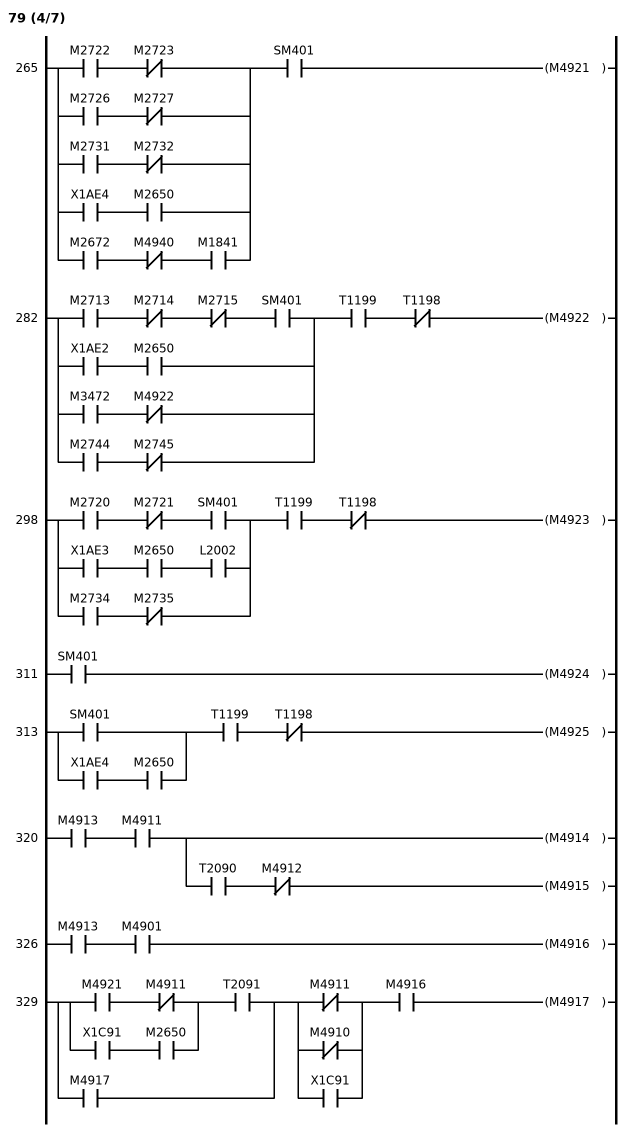
265   LD      M2722
      ANI     M2723
      LD      M2726
      ANI     M2727
      ORB
      LD      M2731
      ANI     M2732
      ORB
      LD      X1AE4
      AND     M2650
      ORB
      LD      M2672
      ANI     M4940
      AND     M1841
      ORB
      AND     SM401
      OUT     M4921
282   LD      M2713
      ANI     M2714
      ANI     M2715
      AND     SM401
      LD      X1AE2
      AND     M2650
      ORB
      LD      M3472
      ANI     M4922
      ORB
      LD      M2744
      ANI     M2745
      ORB
      AND     T1199
      ANI     T1198
      OUT     M4922
298   LD      M2720
      ANI     M2721
      AND     SM401
      LD      X1AE3
      AND     M2650
      AND     L2002
      ORB
      LD      M2734
      ANI     M2735
      ORB
      AND     T1199
      ANI     T1198
      OUT     M4923
311   LD      SM401
      OUT     M4924
313   LD      SM401
      LD      X1AE4
      AND     M2650
      ORB
      AND     T1199
      ANI     T1198
      OUT     M4925
320   LD      M4913
      AND     M4911
      OUT     M4914
      AND     T2090
      ANI     M4912
      OUT     M4915
326   LD      M4913
      AND     M4901
      OUT     M4916
329   LD      M4921
      ANI     M4911
      LD      X1C91
      AND     M2650
      ORB
      AND     T2091
      OR      M4917
      LDI     M4911
      ORI     M4910
      OR      X1C91
      ANB
      AND     M4916
      OUT     M4917
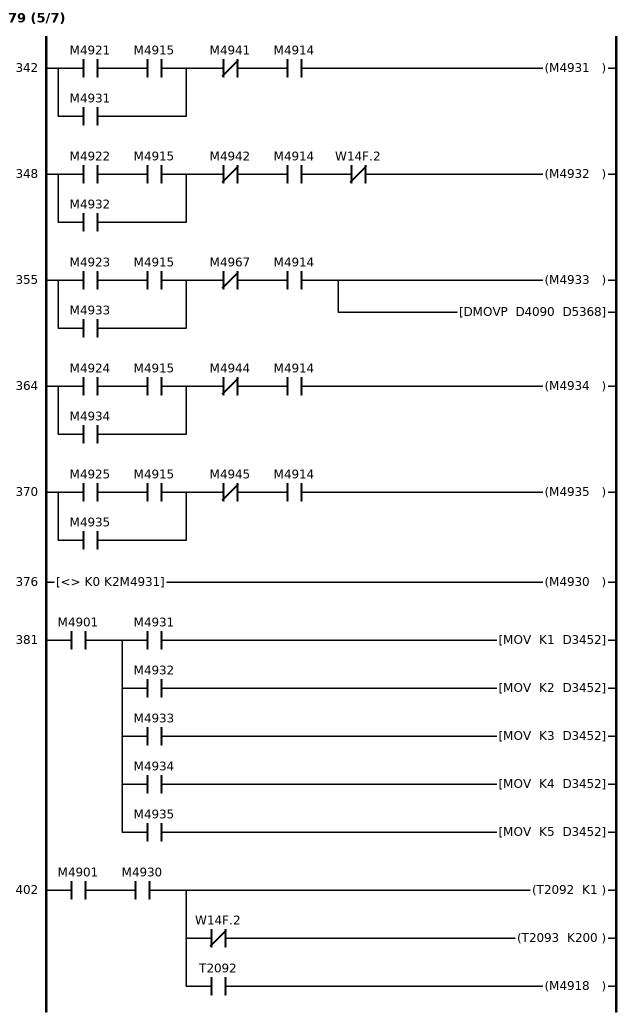
342   LD      M4921
      AND     M4915
      OR      M4931
      ANI     M4941
      AND     M4914
      OUT     M4931
348   LD      M4922
      AND     M4915
      OR      M4932
      ANI     M4942
      AND     M4914
      ANI     W14F.2
      OUT     M4932
355   LD      M4923
      AND     M4915
      OR      M4933
      ANI     M4967
      AND     M4914
      OUT     M4933
      DMOVP   D4090 D5368
364   LD      M4924
      AND     M4915
      OR      M4934
      ANI     M4944
      AND     M4914
      OUT     M4934
370   LD      M4925
      AND     M4915
      OR      M4935
      ANI     M4945
      AND     M4914
      OUT     M4935
376   LD<>    K0 K2M4931
      OUT     M4930
381   LD      M4901
      MPS
      AND     M4931
      MOV     K1 D3452
      MRD
      AND     M4932
      MOV     K2 D3452
      MRD
      AND     M4933
      MOV     K3 D3452
      MRD
      AND     M4934
      MOV     K4 D3452
      MPP
      AND     M4935
      MOV     K5 D3452
402   LD      M4901
      AND     M4930
      OUT     T2092 K1
      MPS
      ANI     W14F.2
      OUT     T2093 K200
      MPP
      AND     T2092
      OUT     M4918
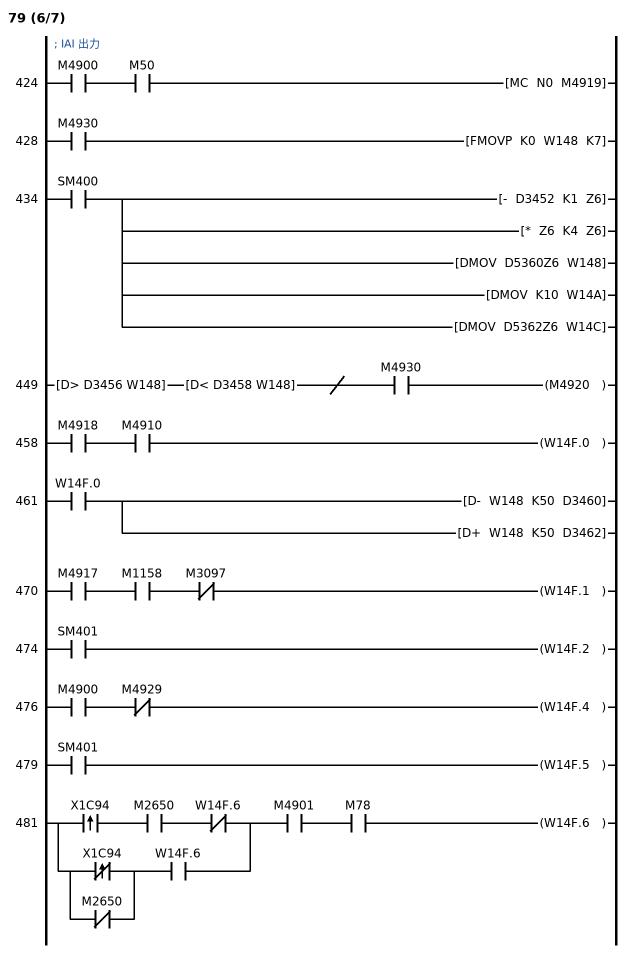
; IAI 出力
424   LD      M4900
      AND     M50
      MC      N0 M4919
428   LD      M4930
      FMOVP   K0 W148 K7
434   LD      SM400
      -       D3452 K1 Z6
      *       Z6 K4 Z6
      DMOV    D5360Z6 W148
      DMOV    K10 W14A
      DMOV    D5362Z6 W14C
449   LDD>    D3456 W148
      ANDD<   D3458 W148
      INV
      AND     M4930
      OUT     M4920
458   LD      M4918
      AND     M4910
      OUT     W14F.0
461   LD      W14F.0
      D-      W148 K50 D3460
      D+      W148 K50 D3462
470   LD      M4917
      AND     M1158
      ANI     M3097
      OUT     W14F.1
474   LD      SM401
      OUT     W14F.2
476   LD      M4900
      ANI     M4929
      OUT     W14F.4
479   LD      SM401
      OUT     W14F.5
481   LDP     X1C94
      AND     M2650
      ANI     W14F.6
      LDPI    X1C94
      ORI     M2650
      AND     W14F.6
      ORB
      AND     M4901
      AND     M78
      OUT     W14F.6
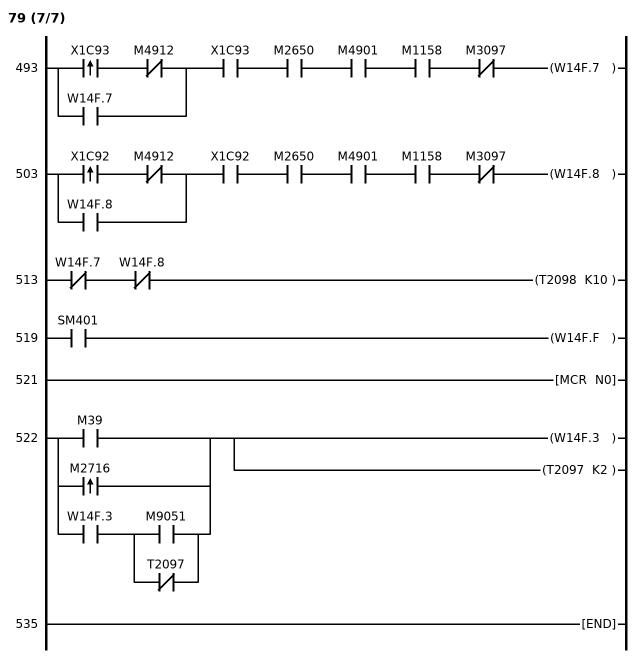
493   LDP     X1C93
      ANI     M4912
      OR      W14F.7
      AND     X1C93
      AND     M2650
      AND     M4901
      AND     M1158
      ANI     M3097
      OUT     W14F.7
503   LDP     X1C92
      ANI     M4912
      OR      W14F.8
      AND     X1C92
      AND     M2650
      AND     M4901
      AND     M1158
      ANI     M3097
      OUT     W14F.8
513   LDI     W14F.7
      ANI     W14F.8
      OUT     T2098 K10
519   LD      SM401
      OUT     W14F.F
521   MCR     N0
522   LD      M39
      ORP     M2716
      LD      W14F.3
      LD      M9051
      ORI     T2097
      ANB
      ORB
      OUT     W14F.3
      OUT     T2097 K2
535   END
END_PROGRAM

PROGRAM 80
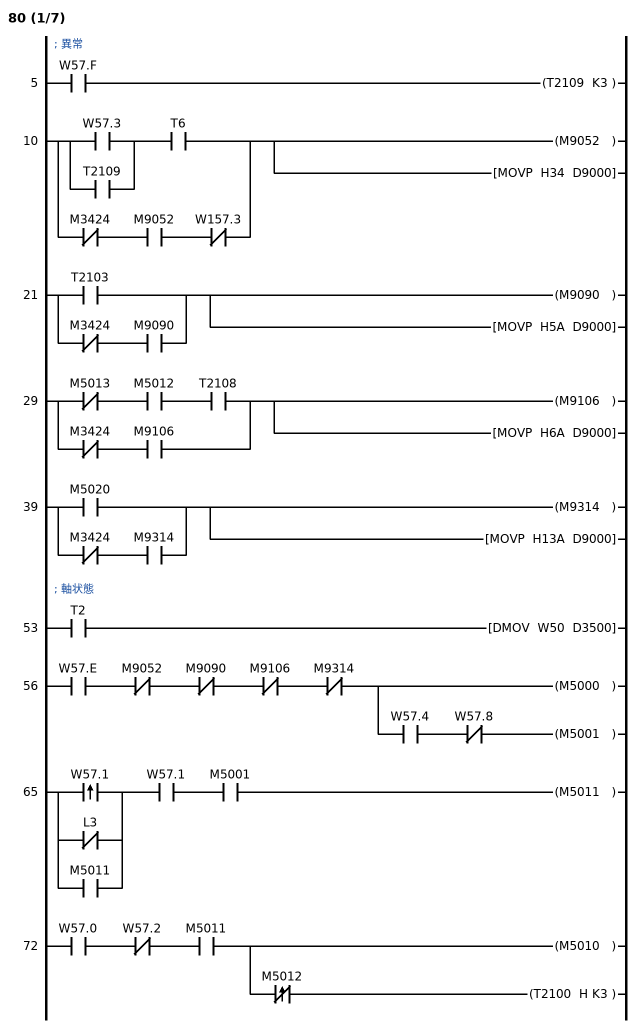
; 異常
5     LD      W57.F
      OUT     T2109 K3
10    LD      W57.3
      OR      T2109
      AND     T6
      LDI     M3424
      AND     M9052
      ANI     W157.3
      ORB
      OUT     M9052
      MOVP    H34 D9000
21    LD      T2103
      LDI     M3424
      AND     M9090
      ORB
      OUT     M9090
      MOVP    H5A D9000
29    LDI     M5013
      AND     M5012
      AND     T2108
      LDI     M3424
      AND     M9106
      ORB
      OUT     M9106
      MOVP    H6A D9000
39    LD      M5020
      LDI     M3424
      AND     M9314
      ORB
      OUT     M9314
      MOVP    H13A D9000
; 軸状態
53    LD      T2
      DMOV    W50 D3500
56    LD      W57.E
      ANI     M9052
      ANI     M9090
      ANI     M9106
      ANI     M9314
      OUT     M5000
      AND     W57.4
      ANI     W57.8
      OUT     M5001
65    LDP     W57.1
      ORI     L3
      OR      M5011
      AND     W57.1
      AND     M5001
      OUT     M5011
72    LD      W57.0
      ANI     W57.2
      AND     M5011
      OUT     M5010
      ANDPI   M5012
      OUTH    T2100 K3
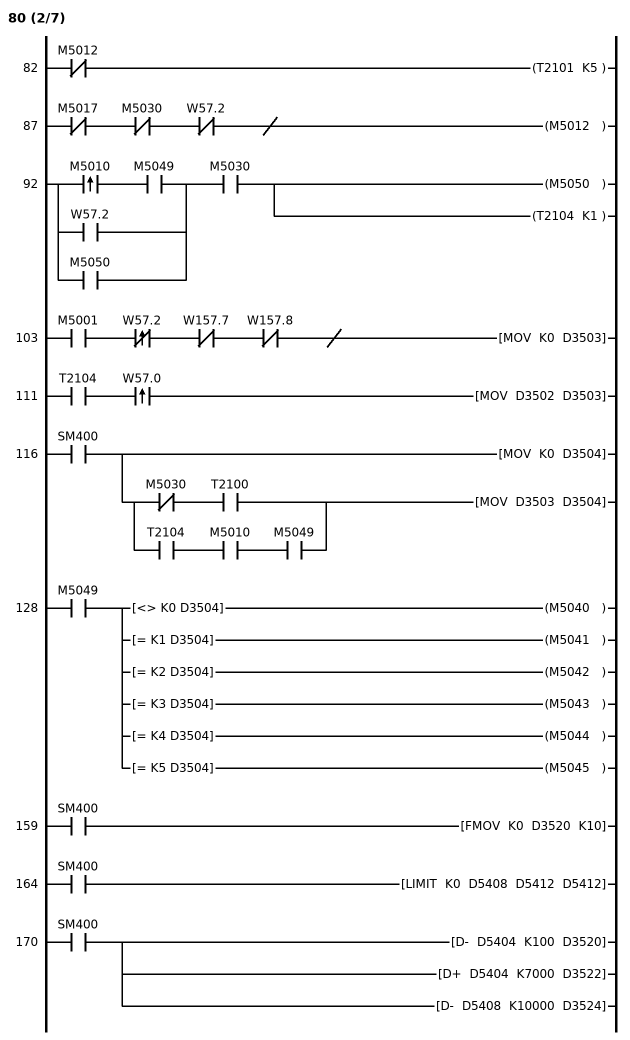
82    LDI     M5012
      OUT     T2101 K5
87    LDI     M5017
      ANI     M5030
      ANI     W57.2
      INV
      OUT     M5012
92    LDP     M5010
      AND     M5049
      OR      W57.2
      OR      M5050
      AND     M5030
      OUT     M5050
      OUT     T2104 K1
103   LD      M5001
      ANDPI   W57.2
      ANI     W157.7
      ANI     W157.8
      INV
      MOV     K0 D3503
111   LD      T2104
      ANDP    W57.0
      MOV     D3502 D3503
116   LD      SM400
      MOV     K0 D3504
      LDI     M5030
      AND     T2100
      LD      T2104
      AND     M5010
      AND     M5049
      ORB
      ANB
      MOV     D3503 D3504
128   LD      M5049
      MPS
      AND<>   K0 D3504
      OUT     M5040
      MRD
      AND=    K1 D3504
      OUT     M5041
      MRD
      AND=    K2 D3504
      OUT     M5042
      MRD
      AND=    K3 D3504
      OUT     M5043
      MRD
      AND=    K4 D3504
      OUT     M5044
      MPP
      AND=    K5 D3504
      OUT     M5045
159   LD      SM400
      FMOV    K0 D3520 K10
164   LD      SM400
      LIMIT   K0 D5408 D5412 D5412
170   LD      SM400
      D-      D5404 K100 D3520
      D+      D5404 K7000 D3522
      D-      D5408 K10000 D3524
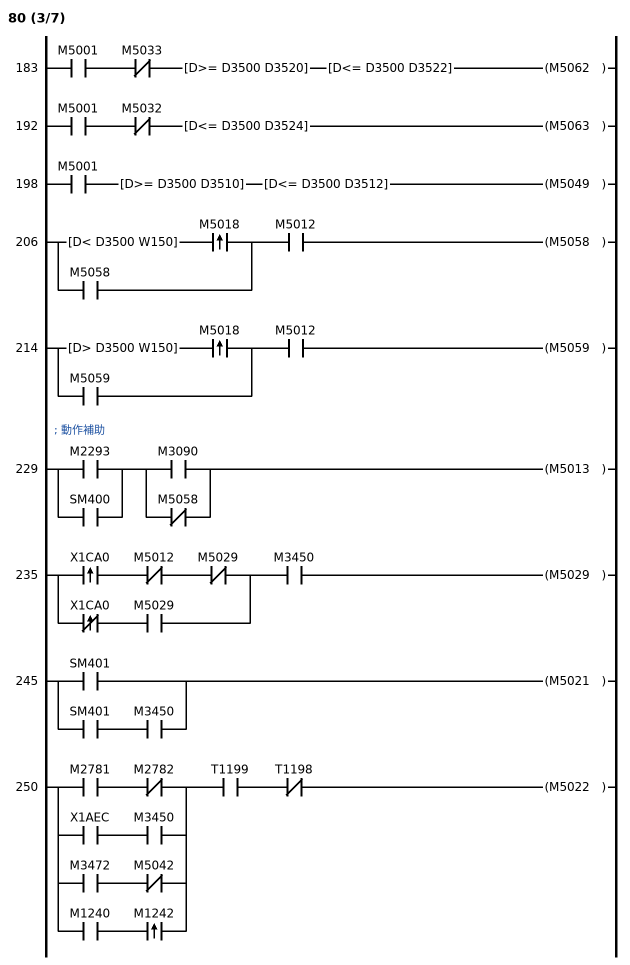
183   LD      M5001
      ANI     M5033
      ANDD>=  D3500 D3520
      ANDD<=  D3500 D3522
      OUT     M5062
192   LD      M5001
      ANI     M5032
      ANDD<=  D3500 D3524
      OUT     M5063
198   LD      M5001
      ANDD>=  D3500 D3510
      ANDD<=  D3500 D3512
      OUT     M5049
206   LDD<    D3500 W150
      ANDP    M5018
      OR      M5058
      AND     M5012
      OUT     M5058
214   LDD>    D3500 W150
      ANDP    M5018
      OR      M5059
      AND     M5012
      OUT     M5059
; 動作補助
229   LD      M2293
      OR      SM400
      LD      M3090
      ORI     M5058
      ANB
      OUT     M5013
235   LDP     X1CA0
      ANI     M5012
      ANI     M5029
      LDPI    X1CA0
      AND     M5029
      ORB
      AND     M3450
      OUT     M5029
245   LD      SM401
      LD      SM401
      AND     M3450
      ORB
      OUT     M5021
250   LD      M2781
      ANI     M2782
      LD      X1AEC
      AND     M3450
      ORB
      LD      M3472
      ANI     M5042
      ORB
      LD      M1240
      ANDP    M1242
      ORB
      AND     T1199
      ANI     T1198
      OUT     M5022
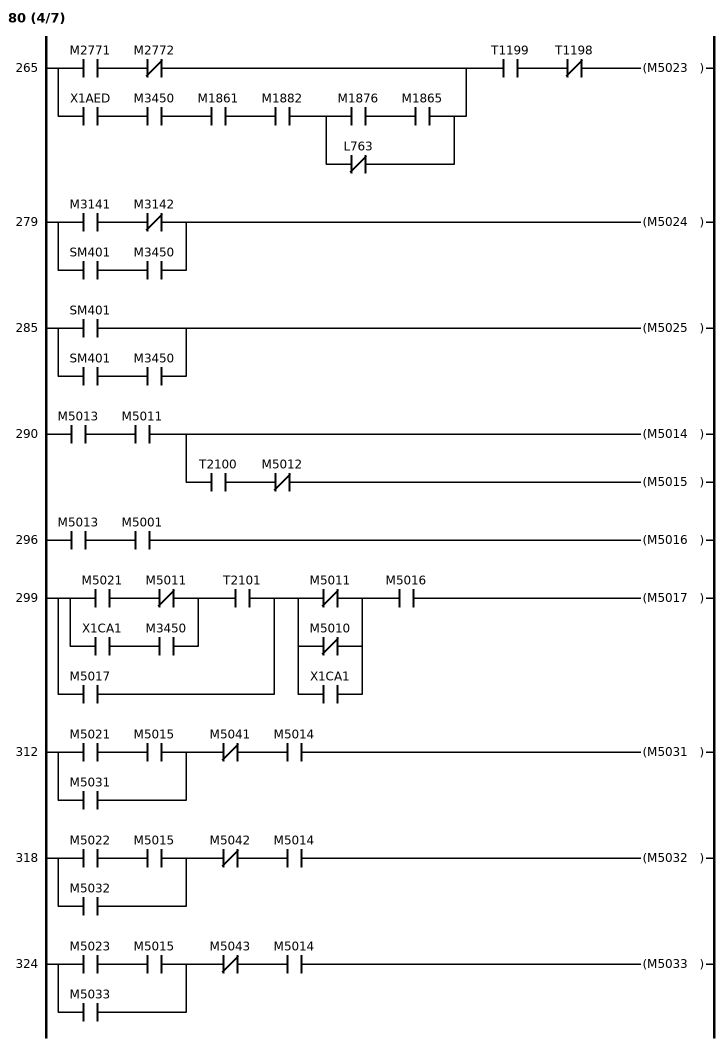
265   LD      M2771
      ANI     M2772
      LD      X1AED
      AND     M3450
      AND     M1861
      AND     M1882
      LD      M1876
      AND     M1865
      ORI     L763
      ANB
      ORB
      AND     T1199
      ANI     T1198
      OUT     M5023
279   LD      M3141
      ANI     M3142
      LD      SM401
      AND     M3450
      ORB
      OUT     M5024
285   LD      SM401
      LD      SM401
      AND     M3450
      ORB
      OUT     M5025
290   LD      M5013
      AND     M5011
      OUT     M5014
      AND     T2100
      ANI     M5012
      OUT     M5015
296   LD      M5013
      AND     M5001
      OUT     M5016
299   LD      M5021
      ANI     M5011
      LD      X1CA1
      AND     M3450
      ORB
      AND     T2101
      OR      M5017
      LDI     M5011
      ORI     M5010
      OR      X1CA1
      ANB
      AND     M5016
      OUT     M5017
312   LD      M5021
      AND     M5015
      OR      M5031
      ANI     M5041
      AND     M5014
      OUT     M5031
318   LD      M5022
      AND     M5015
      OR      M5032
      ANI     M5042
      AND     M5014
      OUT     M5032
324   LD      M5023
      AND     M5015
      OR      M5033
      ANI     M5043
      AND     M5014
      OUT     M5033
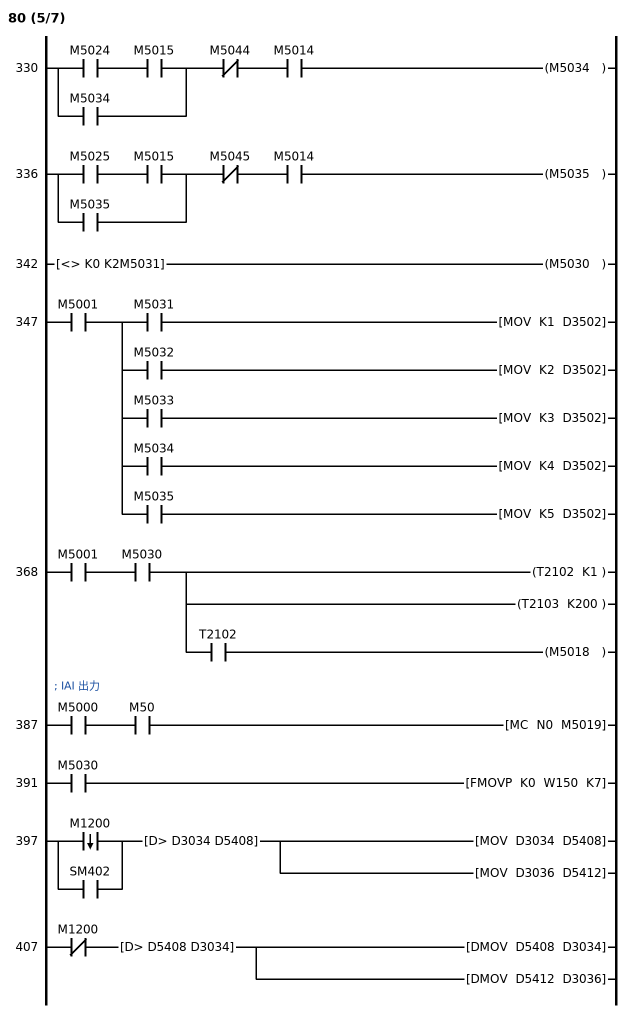
330   LD      M5024
      AND     M5015
      OR      M5034
      ANI     M5044
      AND     M5014
      OUT     M5034
336   LD      M5025
      AND     M5015
      OR      M5035
      ANI     M5045
      AND     M5014
      OUT     M5035
342   LD<>    K0 K2M5031
      OUT     M5030
347   LD      M5001
      MPS
      AND     M5031
      MOV     K1 D3502
      MRD
      AND     M5032
      MOV     K2 D3502
      MRD
      AND     M5033
      MOV     K3 D3502
      MRD
      AND     M5034
      MOV     K4 D3502
      MPP
      AND     M5035
      MOV     K5 D3502
368   LD      M5001
      AND     M5030
      OUT     T2102 K1
      OUT     T2103 K200
      AND     T2102
      OUT     M5018
; IAI 出力
387   LD      M5000
      AND     M50
      MC      N0 M5019
391   LD      M5030
      FMOVP   K0 W150 K7
397   LDF     M1200
      OR      SM402
      ANDD>   D3034 D5408
      MOV     D3034 D5408
      MOV     D3036 D5412
407   LDI     M1200
      ANDD>   D5408 D3034
      DMOV    D5408 D3034
      DMOV    D5412 D3036
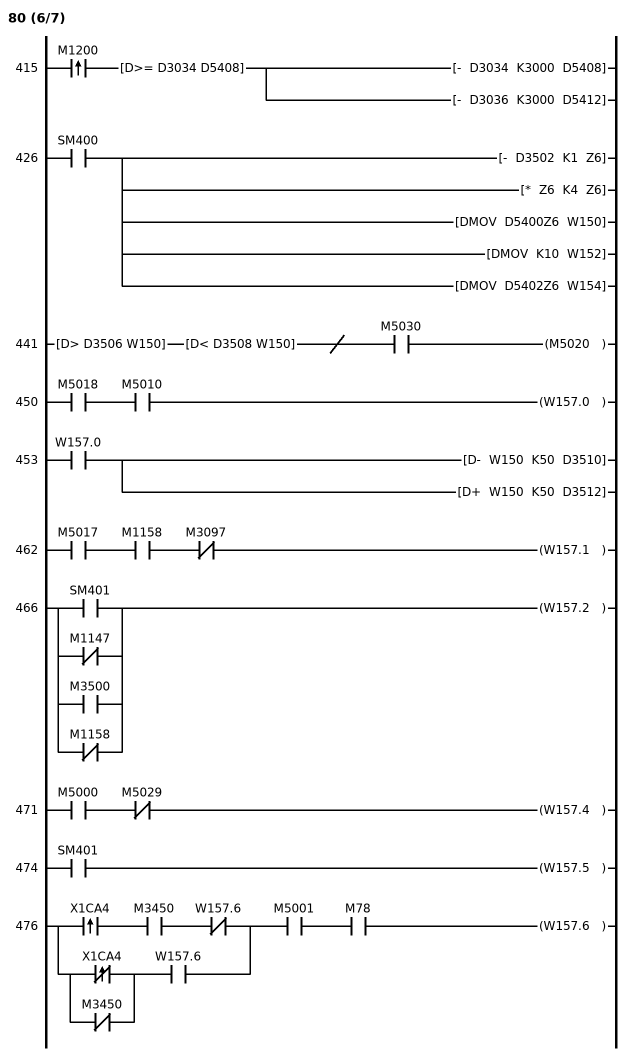
415   LDP     M1200
      ANDD>=  D3034 D5408
      -       D3034 K3000 D5408
      -       D3036 K3000 D5412
426   LD      SM400
      -       D3502 K1 Z6
      *       Z6 K4 Z6
      DMOV    D5400Z6 W150
      DMOV    K10 W152
      DMOV    D5402Z6 W154
441   LDD>    D3506 W150
      ANDD<   D3508 W150
      INV
      AND     M5030
      OUT     M5020
450   LD      M5018
      AND     M5010
      OUT     W157.0
453   LD      W157.0
      D-      W150 K50 D3510
      D+      W150 K50 D3512
462   LD      M5017
      AND     M1158
      ANI     M3097
      OUT     W157.1
466   LD      SM401
      ORI     M1147
      OR      M3500
      ORI     M1158
      OUT     W157.2
471   LD      M5000
      ANI     M5029
      OUT     W157.4
474   LD      SM401
      OUT     W157.5
476   LDP     X1CA4
      AND     M3450
      ANI     W157.6
      LDPI    X1CA4
      ORI     M3450
      AND     W157.6
      ORB
      AND     M5001
      AND     M78
      OUT     W157.6
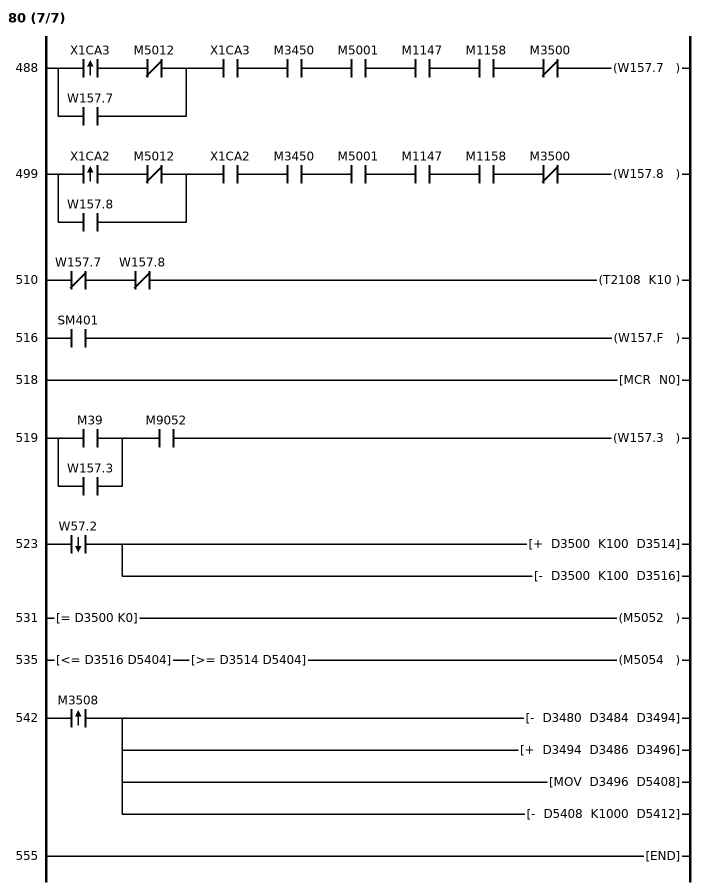
488   LDP     X1CA3
      ANI     M5012
      OR      W157.7
      AND     X1CA3
      AND     M3450
      AND     M5001
      AND     M1147
      AND     M1158
      ANI     M3500
      OUT     W157.7
499   LDP     X1CA2
      ANI     M5012
      OR      W157.8
      AND     X1CA2
      AND     M3450
      AND     M5001
      AND     M1147
      AND     M1158
      ANI     M3500
      OUT     W157.8
510   LDI     W157.7
      ANI     W157.8
      OUT     T2108 K10
516   LD      SM401
      OUT     W157.F
518   MCR     N0
519   LD      M39
      OR      W157.3
      AND     M9052
      OUT     W157.3
523   LDF     W57.2
      +       D3500 K100 D3514
      -       D3500 K100 D3516
531   LD=     D3500 K0
      OUT     M5052
535   LD<=    D3516 D5404
      AND>=   D3514 D5404
      OUT     M5054
542   LDP     M3508
      -       D3480 D3484 D3494
      +       D3494 D3486 D3496
      MOV     D3496 D5408
      -       D5408 K1000 D5412
555   END
END_PROGRAM

PROGRAM 81
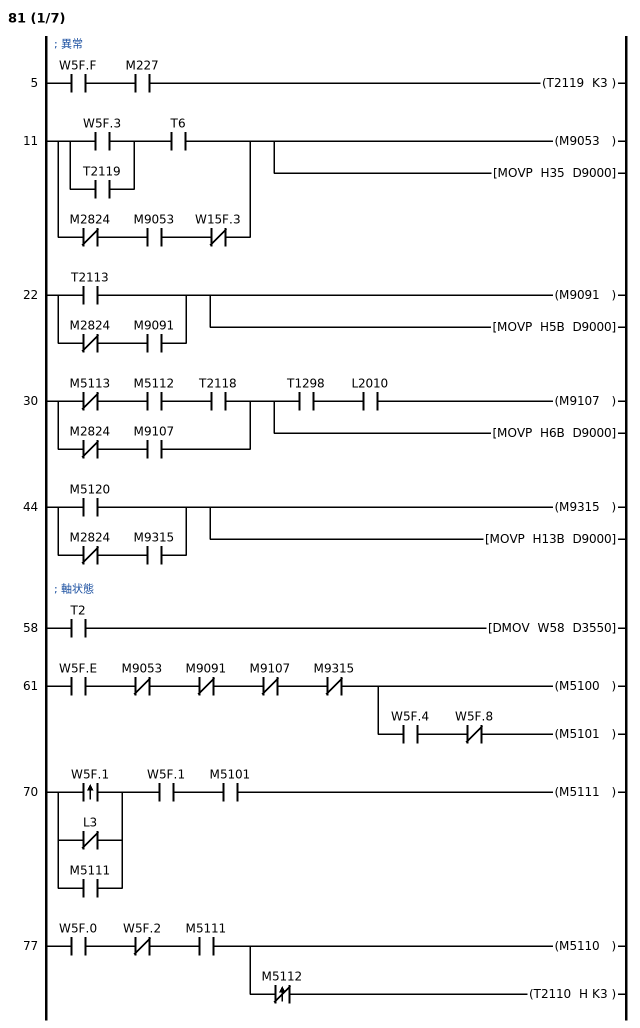
; 異常
5     LD      W5F.F
      AND     M227
      OUT     T2119 K3
11    LD      W5F.3
      OR      T2119
      AND     T6
      LDI     M2824
      AND     M9053
      ANI     W15F.3
      ORB
      OUT     M9053
      MOVP    H35 D9000
22    LD      T2113
      LDI     M2824
      AND     M9091
      ORB
      OUT     M9091
      MOVP    H5B D9000
30    LDI     M5113
      AND     M5112
      AND     T2118
      LDI     M2824
      AND     M9107
      ORB
      MPS
      AND     T1298
      AND     L2010
      OUT     M9107
      MPP
      MOVP    H6B D9000
44    LD      M5120
      LDI     M2824
      AND     M9315
      ORB
      OUT     M9315
      MOVP    H13B D9000
; 軸状態
58    LD      T2
      DMOV    W58 D3550
61    LD      W5F.E
      ANI     M9053
      ANI     M9091
      ANI     M9107
      ANI     M9315
      OUT     M5100
      AND     W5F.4
      ANI     W5F.8
      OUT     M5101
70    LDP     W5F.1
      ORI     L3
      OR      M5111
      AND     W5F.1
      AND     M5101
      OUT     M5111
77    LD      W5F.0
      ANI     W5F.2
      AND     M5111
      OUT     M5110
      ANDPI   M5112
      OUTH    T2110 K3
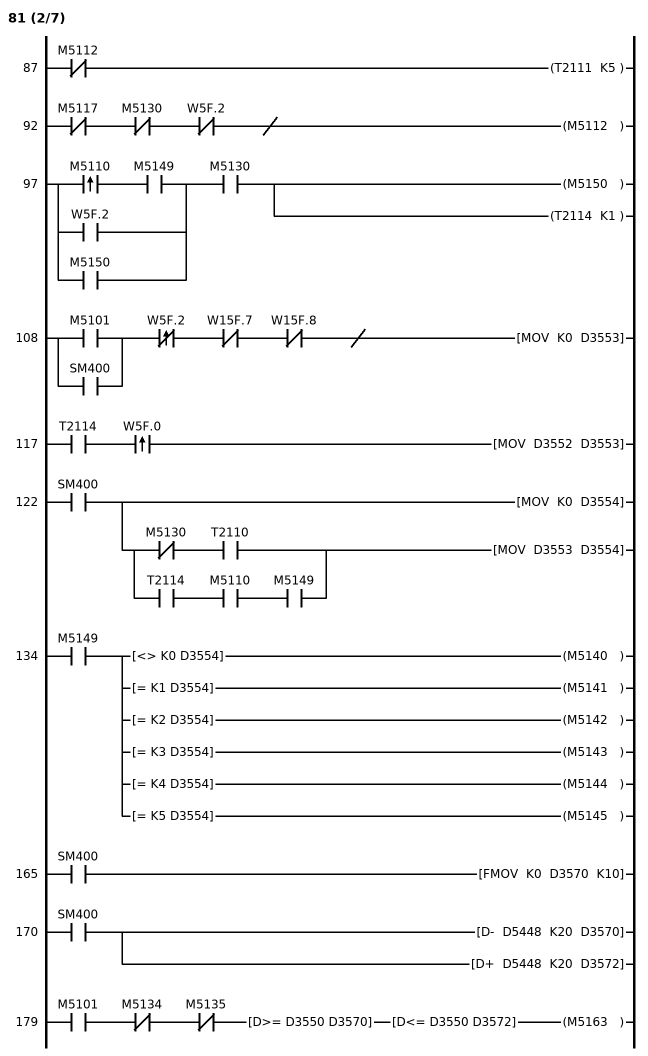
87    LDI     M5112
      OUT     T2111 K5
92    LDI     M5117
      ANI     M5130
      ANI     W5F.2
      INV
      OUT     M5112
97    LDP     M5110
      AND     M5149
      OR      W5F.2
      OR      M5150
      AND     M5130
      OUT     M5150
      OUT     T2114 K1
108   LD      M5101
      OR      SM400
      ANDPI   W5F.2
      ANI     W15F.7
      ANI     W15F.8
      INV
      MOV     K0 D3553
117   LD      T2114
      ANDP    W5F.0
      MOV     D3552 D3553
122   LD      SM400
      MOV     K0 D3554
      LDI     M5130
      AND     T2110
      LD      T2114
      AND     M5110
      AND     M5149
      ORB
      ANB
      MOV     D3553 D3554
134   LD      M5149
      MPS
      AND<>   K0 D3554
      OUT     M5140
      MRD
      AND=    K1 D3554
      OUT     M5141
      MRD
      AND=    K2 D3554
      OUT     M5142
      MRD
      AND=    K3 D3554
      OUT     M5143
      MRD
      AND=    K4 D3554
      OUT     M5144
      MPP
      AND=    K5 D3554
      OUT     M5145
165   LD      SM400
      FMOV    K0 D3570 K10
170   LD      SM400
      D-      D5448 K20 D3570
      D+      D5448 K20 D3572
179   LD      M5101
      ANI     M5134
      ANI     M5135
      ANDD>=  D3550 D3570
      ANDD<=  D3550 D3572
      OUT     M5163
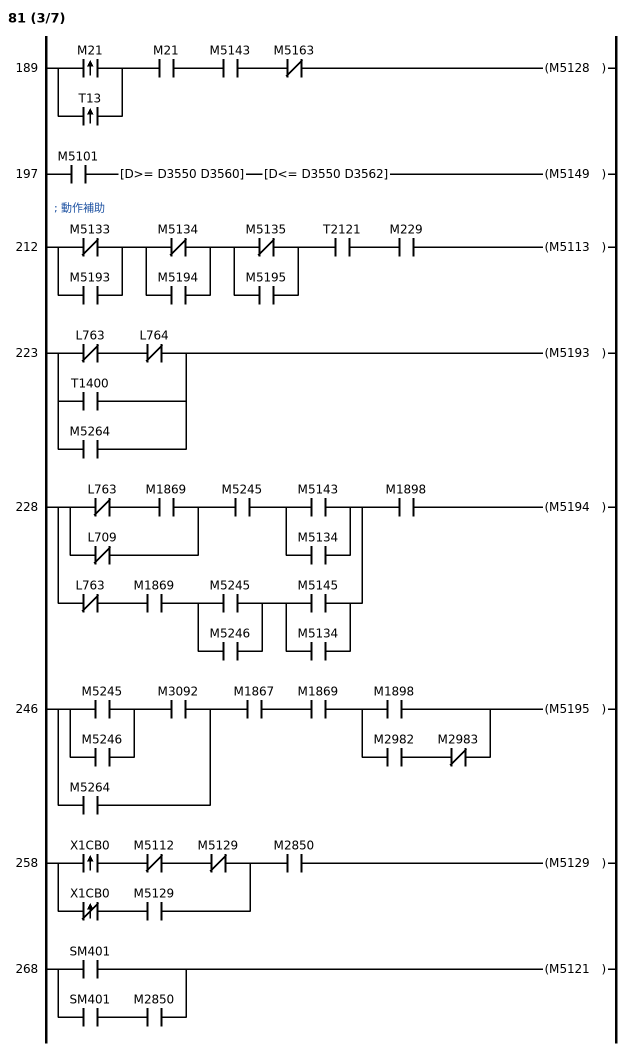
189   LDP     M21
      ORP     T13
      AND     M21
      AND     M5143
      ANI     M5163
      OUT     M5128
197   LD      M5101
      ANDD>=  D3550 D3560
      ANDD<=  D3550 D3562
      OUT     M5149
; 動作補助
212   LDI     M5133
      OR      M5193
      LDI     M5134
      OR      M5194
      ANB
      LDI     M5135
      OR      M5195
      ANB
      AND     T2121
      AND     M229
      OUT     M5113
223   LDI     L763
      ANI     L764
      OR      T1400
      OR      M5264
      OUT     M5193
228   LDI     L763
      AND     M1869
      ORI     L709
      AND     M5245
      LD      M5143
      OR      M5134
      ANB
      LDI     L763
      AND     M1869
      LD      M5245
      OR      M5246
      ANB
      LD      M5145
      OR      M5134
      ANB
      ORB
      AND     M1898
      OUT     M5194
246   LD      M5245
      OR      M5246
      AND     M3092
      OR      M5264
      AND     M1867
      AND     M1869
      LD      M1898
      LD      M2982
      ANI     M2983
      ORB
      ANB
      OUT     M5195
258   LDP     X1CB0
      ANI     M5112
      ANI     M5129
      LDPI    X1CB0
      AND     M5129
      ORB
      AND     M2850
      OUT     M5129
268   LD      SM401
      LD      SM401
      AND     M2850
      ORB
      OUT     M5121
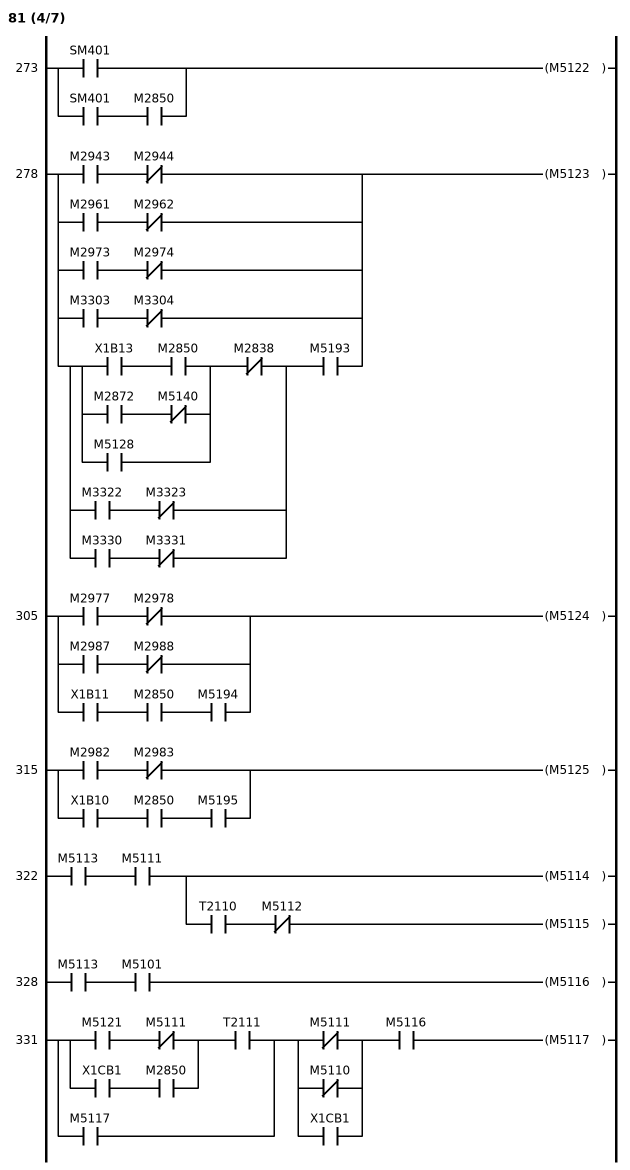
273   LD      SM401
      LD      SM401
      AND     M2850
      ORB
      OUT     M5122
278   LD      M2943
      ANI     M2944
      LD      M2961
      ANI     M2962
      ORB
      LD      M2973
      ANI     M2974
      ORB
      LD      M3303
      ANI     M3304
      ORB
      LD      X1B13
      AND     M2850
      LD      M2872
      ANI     M5140
      ORB
      OR      M5128
      ANI     M2838
      LD      M3322
      ANI     M3323
      ORB
      LD      M3330
      ANI     M3331
      ORB
      AND     M5193
      ORB
      OUT     M5123
305   LD      M2977
      ANI     M2978
      LD      M2987
      ANI     M2988
      ORB
      LD      X1B11
      AND     M2850
      AND     M5194
      ORB
      OUT     M5124
315   LD      M2982
      ANI     M2983
      LD      X1B10
      AND     M2850
      AND     M5195
      ORB
      OUT     M5125
322   LD      M5113
      AND     M5111
      OUT     M5114
      AND     T2110
      ANI     M5112
      OUT     M5115
328   LD      M5113
      AND     M5101
      OUT     M5116
331   LD      M5121
      ANI     M5111
      LD      X1CB1
      AND     M2850
      ORB
      AND     T2111
      OR      M5117
      LDI     M5111
      ORI     M5110
      OR      X1CB1
      ANB
      AND     M5116
      OUT     M5117
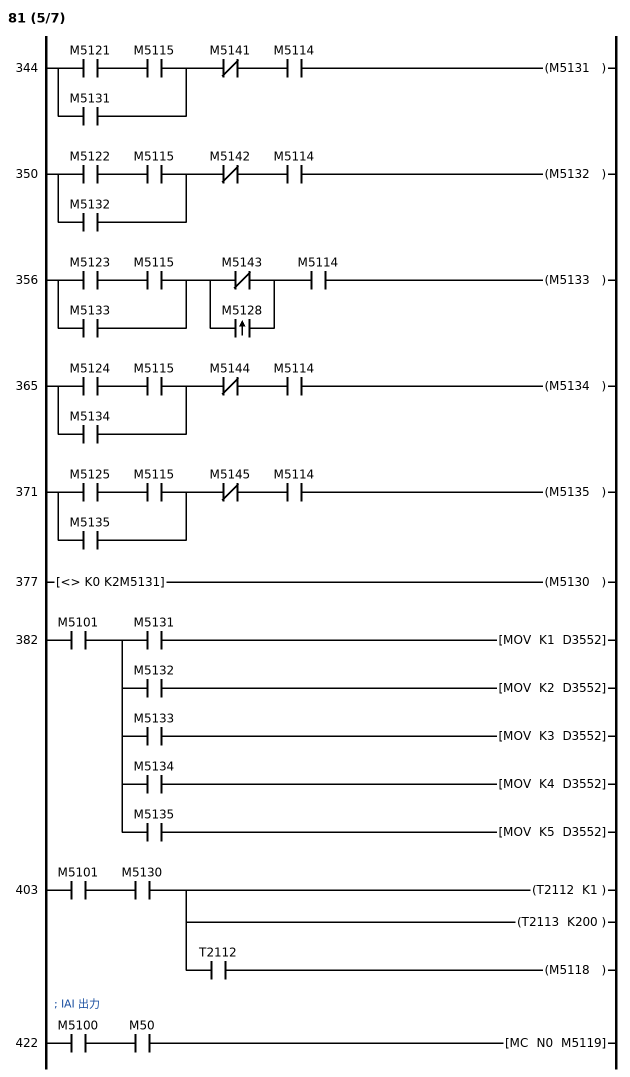
344   LD      M5121
      AND     M5115
      OR      M5131
      ANI     M5141
      AND     M5114
      OUT     M5131
350   LD      M5122
      AND     M5115
      OR      M5132
      ANI     M5142
      AND     M5114
      OUT     M5132
356   LD      M5123
      AND     M5115
      OR      M5133
      LDI     M5143
      ORP     M5128
      ANB
      AND     M5114
      OUT     M5133
365   LD      M5124
      AND     M5115
      OR      M5134
      ANI     M5144
      AND     M5114
      OUT     M5134
371   LD      M5125
      AND     M5115
      OR      M5135
      ANI     M5145
      AND     M5114
      OUT     M5135
377   LD<>    K0 K2M5131
      OUT     M5130
382   LD      M5101
      MPS
      AND     M5131
      MOV     K1 D3552
      MRD
      AND     M5132
      MOV     K2 D3552
      MRD
      AND     M5133
      MOV     K3 D3552
      MRD
      AND     M5134
      MOV     K4 D3552
      MPP
      AND     M5135
      MOV     K5 D3552
403   LD      M5101
      AND     M5130
      OUT     T2112 K1
      OUT     T2113 K200
      AND     T2112
      OUT     M5118
; IAI 出力
422   LD      M5100
      AND     M50
      MC      N0 M5119
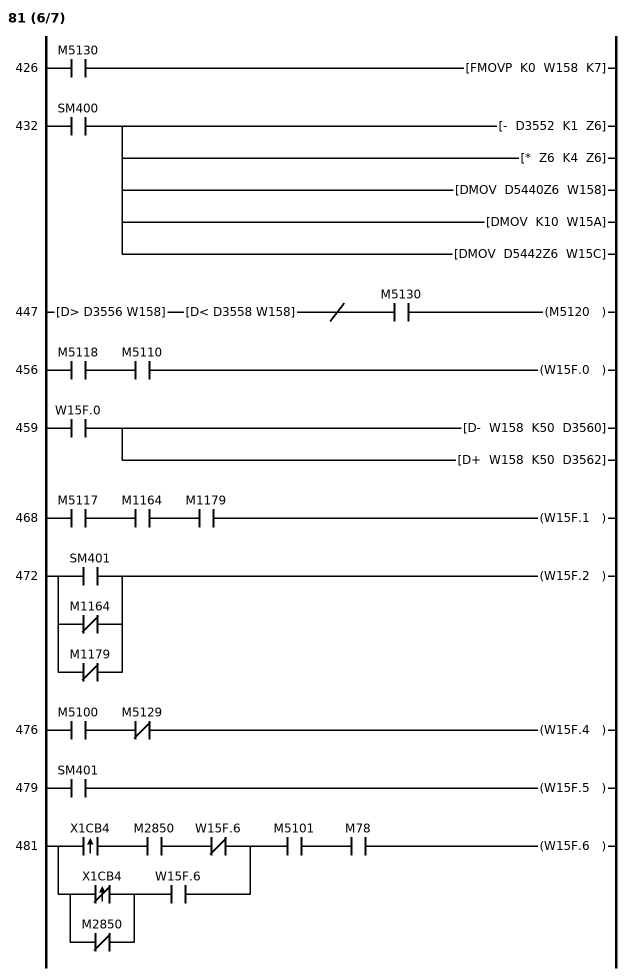
426   LD      M5130
      FMOVP   K0 W158 K7
432   LD      SM400
      -       D3552 K1 Z6
      *       Z6 K4 Z6
      DMOV    D5440Z6 W158
      DMOV    K10 W15A
      DMOV    D5442Z6 W15C
447   LDD>    D3556 W158
      ANDD<   D3558 W158
      INV
      AND     M5130
      OUT     M5120
456   LD      M5118
      AND     M5110
      OUT     W15F.0
459   LD      W15F.0
      D-      W158 K50 D3560
      D+      W158 K50 D3562
468   LD      M5117
      AND     M1164
      AND     M1179
      OUT     W15F.1
472   LD      SM401
      ORI     M1164
      ORI     M1179
      OUT     W15F.2
476   LD      M5100
      ANI     M5129
      OUT     W15F.4
479   LD      SM401
      OUT     W15F.5
481   LDP     X1CB4
      AND     M2850
      ANI     W15F.6
      LDPI    X1CB4
      ORI     M2850
      AND     W15F.6
      ORB
      AND     M5101
      AND     M78
      OUT     W15F.6
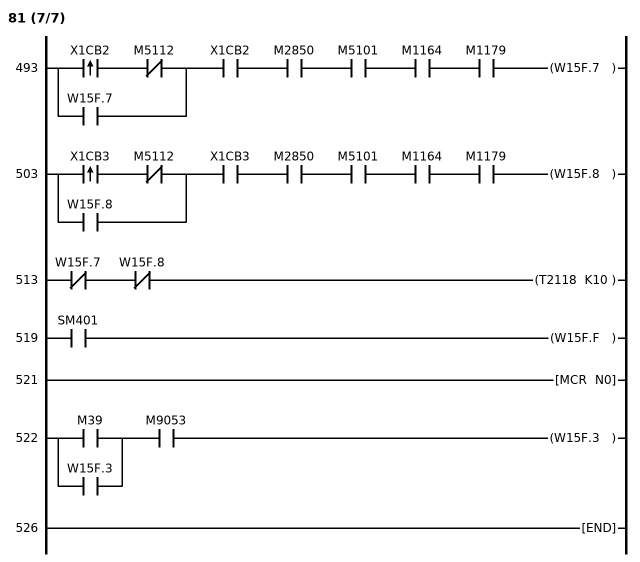
493   LDP     X1CB2
      ANI     M5112
      OR      W15F.7
      AND     X1CB2
      AND     M2850
      AND     M5101
      AND     M1164
      AND     M1179
      OUT     W15F.7
503   LDP     X1CB3
      ANI     M5112
      OR      W15F.8
      AND     X1CB3
      AND     M2850
      AND     M5101
      AND     M1164
      AND     M1179
      OUT     W15F.8
513   LDI     W15F.7
      ANI     W15F.8
      OUT     T2118 K10
519   LD      SM401
      OUT     W15F.F
521   MCR     N0
522   LD      M39
      OR      W15F.3
      AND     M9053
      OUT     W15F.3
526   END
END_PROGRAM

PROGRAM 82
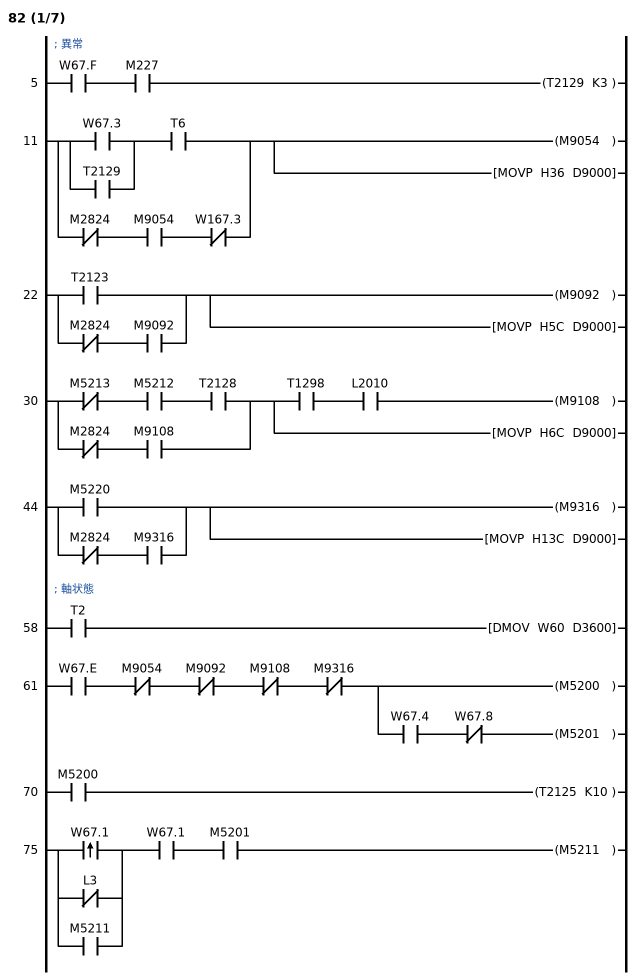
; 異常
5     LD      W67.F
      AND     M227
      OUT     T2129 K3
11    LD      W67.3
      OR      T2129
      AND     T6
      LDI     M2824
      AND     M9054
      ANI     W167.3
      ORB
      OUT     M9054
      MOVP    H36 D9000
22    LD      T2123
      LDI     M2824
      AND     M9092
      ORB
      OUT     M9092
      MOVP    H5C D9000
30    LDI     M5213
      AND     M5212
      AND     T2128
      LDI     M2824
      AND     M9108
      ORB
      MPS
      AND     T1298
      AND     L2010
      OUT     M9108
      MPP
      MOVP    H6C D9000
44    LD      M5220
      LDI     M2824
      AND     M9316
      ORB
      OUT     M9316
      MOVP    H13C D9000
; 軸状態
58    LD      T2
      DMOV    W60 D3600
61    LD      W67.E
      ANI     M9054
      ANI     M9092
      ANI     M9108
      ANI     M9316
      OUT     M5200
      AND     W67.4
      ANI     W67.8
      OUT     M5201
70    LD      M5200
      OUT     T2125 K10
75    LDP     W67.1
      ORI     L3
      OR      M5211
      AND     W67.1
      AND     M5201
      OUT     M5211
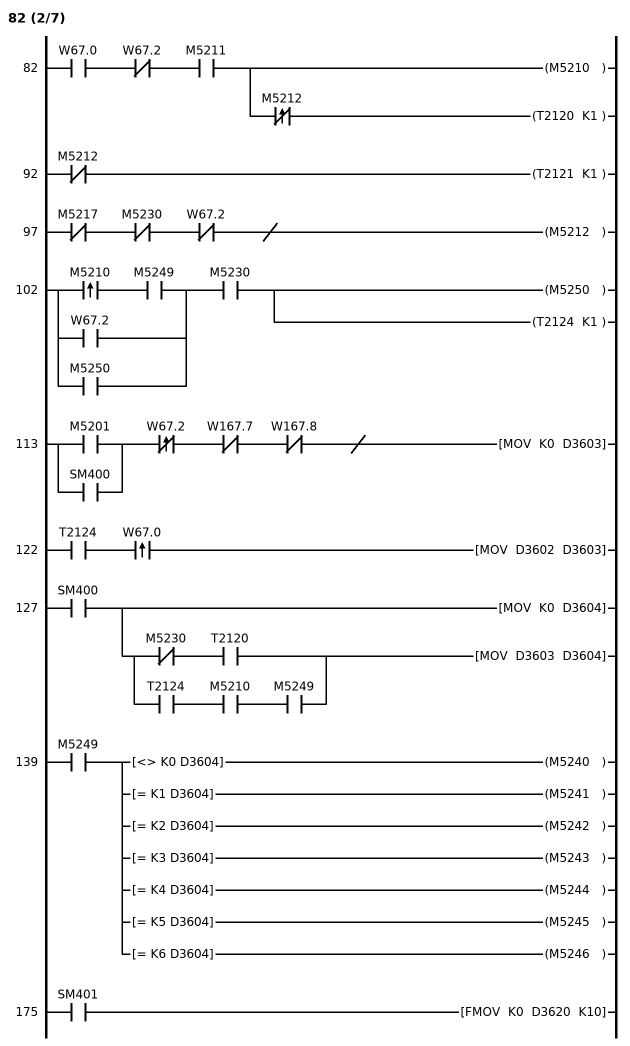
82    LD      W67.0
      ANI     W67.2
      AND     M5211
      OUT     M5210
      ANDPI   M5212
      OUT     T2120 K1
92    LDI     M5212
      OUT     T2121 K1
97    LDI     M5217
      ANI     M5230
      ANI     W67.2
      INV
      OUT     M5212
102   LDP     M5210
      AND     M5249
      OR      W67.2
      OR      M5250
      AND     M5230
      OUT     M5250
      OUT     T2124 K1
113   LD      M5201
      OR      SM400
      ANDPI   W67.2
      ANI     W167.7
      ANI     W167.8
      INV
      MOV     K0 D3603
122   LD      T2124
      ANDP    W67.0
      MOV     D3602 D3603
127   LD      SM400
      MOV     K0 D3604
      LDI     M5230
      AND     T2120
      LD      T2124
      AND     M5210
      AND     M5249
      ORB
      ANB
      MOV     D3603 D3604
139   LD      M5249
      MPS
      AND<>   K0 D3604
      OUT     M5240
      MRD
      AND=    K1 D3604
      OUT     M5241
      MRD
      AND=    K2 D3604
      OUT     M5242
      MRD
      AND=    K3 D3604
      OUT     M5243
      MRD
      AND=    K4 D3604
      OUT     M5244
      MRD
      AND=    K5 D3604
      OUT     M5245
      MPP
      AND=    K6 D3604
      OUT     M5246
175   LD      SM401
      FMOV    K0 D3620 K10
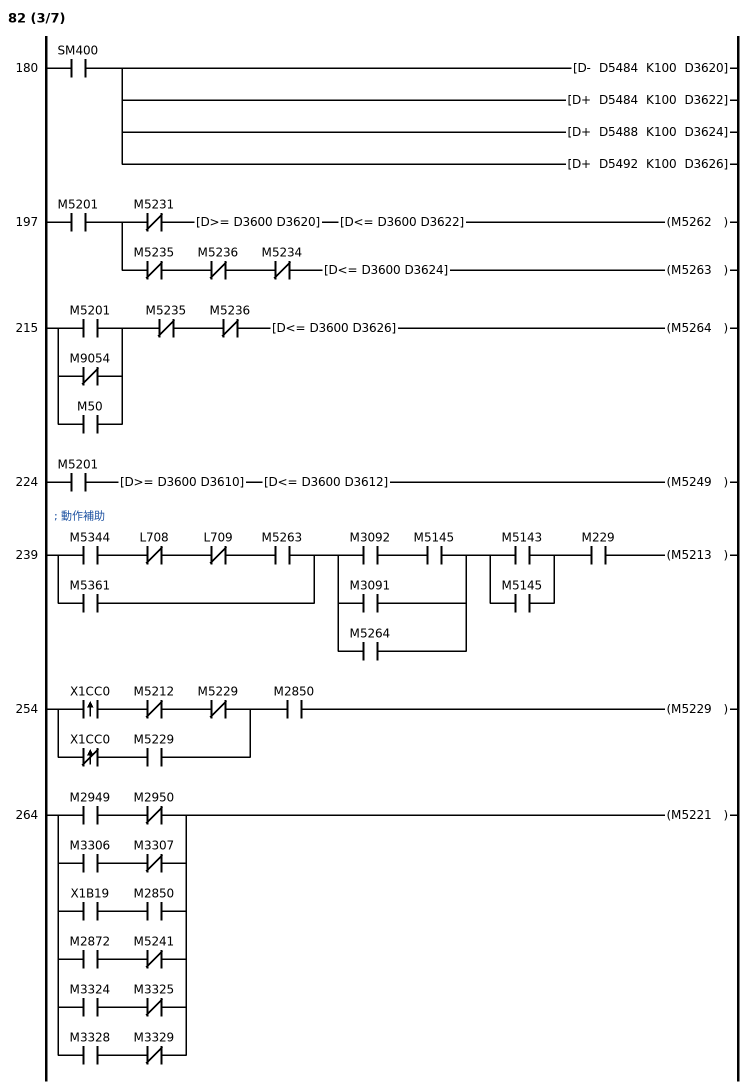
180   LD      SM400
      D-      D5484 K100 D3620
      D+      D5484 K100 D3622
      D+      D5488 K100 D3624
      D+      D5492 K100 D3626
197   LD      M5201
      MPS
      ANI     M5231
      ANDD>=  D3600 D3620
      ANDD<=  D3600 D3622
      OUT     M5262
      MPP
      ANI     M5235
      ANI     M5236
      ANI     M5234
      ANDD<=  D3600 D3624
      OUT     M5263
215   LD      M5201
      ORI     M9054
      OR      M50
      ANI     M5235
      ANI     M5236
      ANDD<=  D3600 D3626
      OUT     M5264
224   LD      M5201
      ANDD>=  D3600 D3610
      ANDD<=  D3600 D3612
      OUT     M5249
; 動作補助
239   LD      M5344
      ANI     L708
      ANI     L709
      AND     M5263
      OR      M5361
      LD      M3092
      AND     M5145
      OR      M3091
      OR      M5264
      ANB
      LD      M5143
      OR      M5145
      ANB
      AND     M229
      OUT     M5213
254   LDP     X1CC0
      ANI     M5212
      ANI     M5229
      LDPI    X1CC0
      AND     M5229
      ORB
      AND     M2850
      OUT     M5229
264   LD      M2949
      ANI     M2950
      LD      M3306
      ANI     M3307
      ORB
      LD      X1B19
      AND     M2850
      ORB
      LD      M2872
      ANI     M5241
      ORB
      LD      M3324
      ANI     M3325
      ORB
      LD      M3328
      ANI     M3329
      ORB
      OUT     M5221
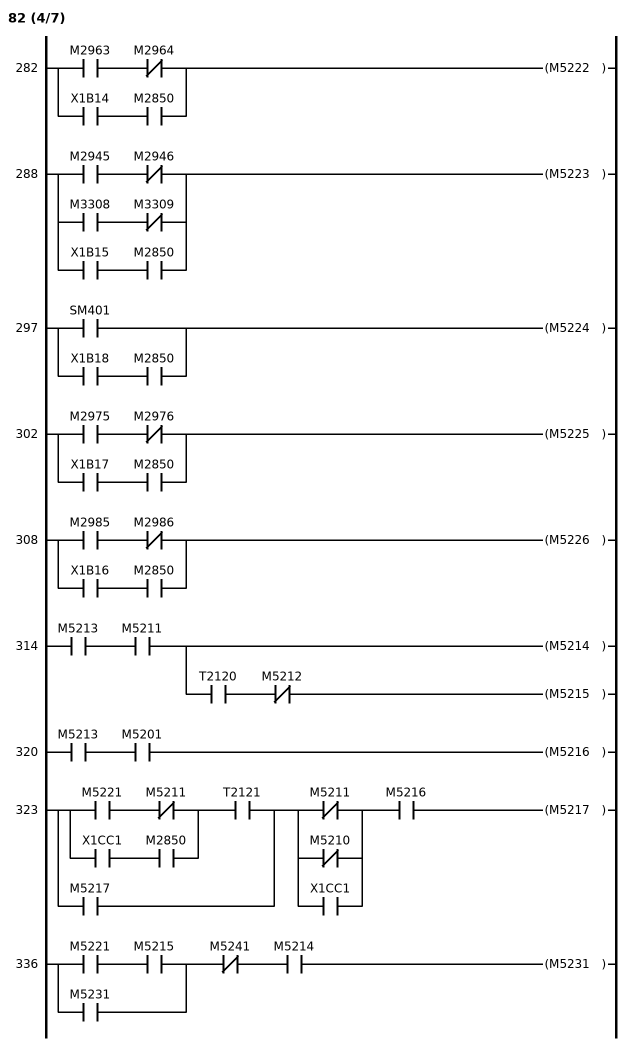
282   LD      M2963
      ANI     M2964
      LD      X1B14
      AND     M2850
      ORB
      OUT     M5222
288   LD      M2945
      ANI     M2946
      LD      M3308
      ANI     M3309
      ORB
      LD      X1B15
      AND     M2850
      ORB
      OUT     M5223
297   LD      SM401
      LD      X1B18
      AND     M2850
      ORB
      OUT     M5224
302   LD      M2975
      ANI     M2976
      LD      X1B17
      AND     M2850
      ORB
      OUT     M5225
308   LD      M2985
      ANI     M2986
      LD      X1B16
      AND     M2850
      ORB
      OUT     M5226
314   LD      M5213
      AND     M5211
      OUT     M5214
      AND     T2120
      ANI     M5212
      OUT     M5215
320   LD      M5213
      AND     M5201
      OUT     M5216
323   LD      M5221
      ANI     M5211
      LD      X1CC1
      AND     M2850
      ORB
      AND     T2121
      OR      M5217
      LDI     M5211
      ORI     M5210
      OR      X1CC1
      ANB
      AND     M5216
      OUT     M5217
336   LD      M5221
      AND     M5215
      OR      M5231
      ANI     M5241
      AND     M5214
      OUT     M5231
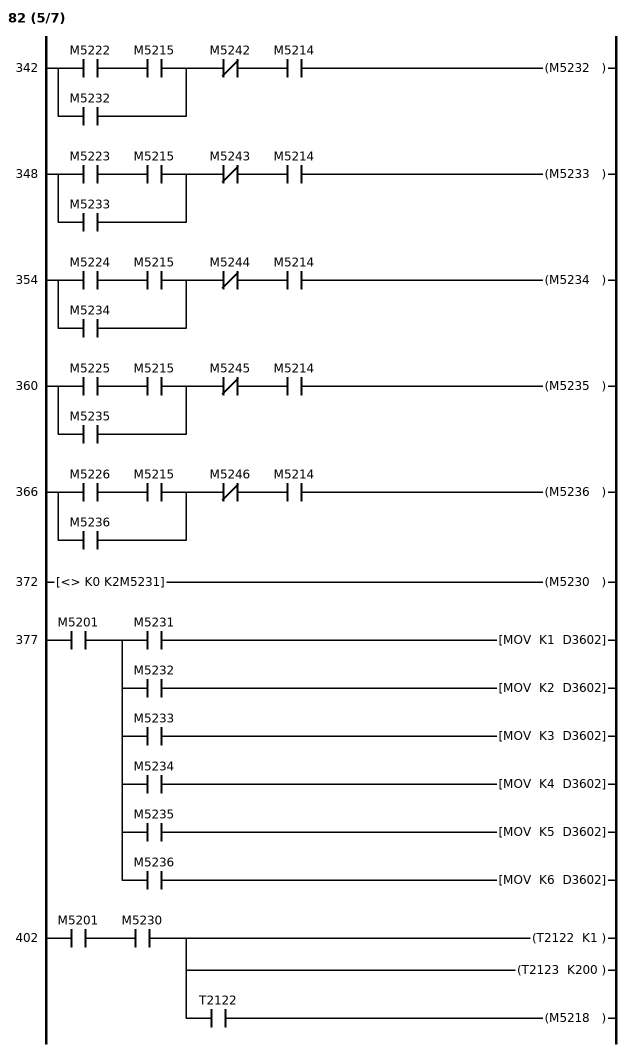
342   LD      M5222
      AND     M5215
      OR      M5232
      ANI     M5242
      AND     M5214
      OUT     M5232
348   LD      M5223
      AND     M5215
      OR      M5233
      ANI     M5243
      AND     M5214
      OUT     M5233
354   LD      M5224
      AND     M5215
      OR      M5234
      ANI     M5244
      AND     M5214
      OUT     M5234
360   LD      M5225
      AND     M5215
      OR      M5235
      ANI     M5245
      AND     M5214
      OUT     M5235
366   LD      M5226
      AND     M5215
      OR      M5236
      ANI     M5246
      AND     M5214
      OUT     M5236
372   LD<>    K0 K2M5231
      OUT     M5230
377   LD      M5201
      MPS
      AND     M5231
      MOV     K1 D3602
      MRD
      AND     M5232
      MOV     K2 D3602
      MRD
      AND     M5233
      MOV     K3 D3602
      MRD
      AND     M5234
      MOV     K4 D3602
      MRD
      AND     M5235
      MOV     K5 D3602
      MPP
      AND     M5236
      MOV     K6 D3602
402   LD      M5201
      AND     M5230
      OUT     T2122 K1
      OUT     T2123 K200
      AND     T2122
      OUT     M5218
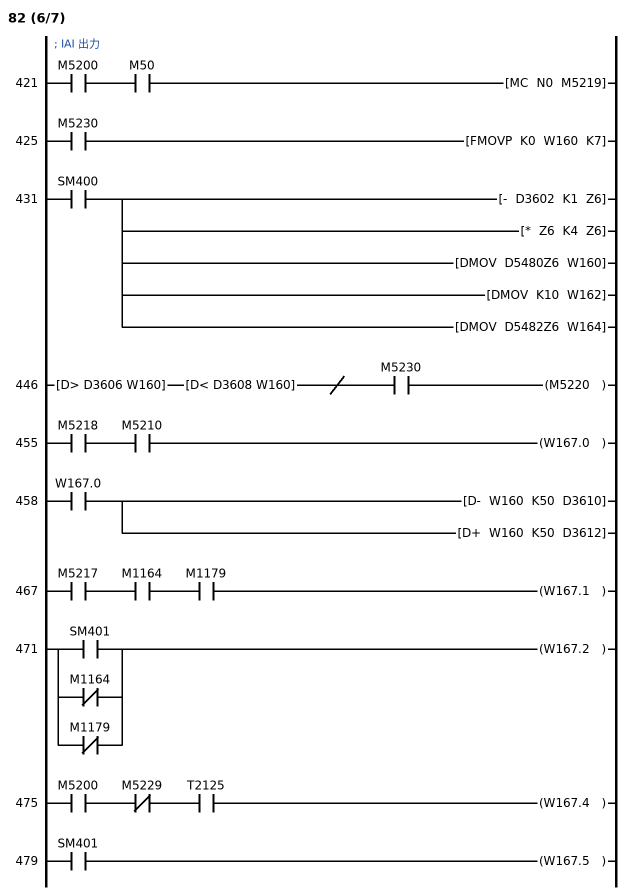
; IAI 出力
421   LD      M5200
      AND     M50
      MC      N0 M5219
425   LD      M5230
      FMOVP   K0 W160 K7
431   LD      SM400
      -       D3602 K1 Z6
      *       Z6 K4 Z6
      DMOV    D5480Z6 W160
      DMOV    K10 W162
      DMOV    D5482Z6 W164
446   LDD>    D3606 W160
      ANDD<   D3608 W160
      INV
      AND     M5230
      OUT     M5220
455   LD      M5218
      AND     M5210
      OUT     W167.0
458   LD      W167.0
      D-      W160 K50 D3610
      D+      W160 K50 D3612
467   LD      M5217
      AND     M1164
      AND     M1179
      OUT     W167.1
471   LD      SM401
      ORI     M1164
      ORI     M1179
      OUT     W167.2
475   LD      M5200
      ANI     M5229
      AND     T2125
      OUT     W167.4
479   LD      SM401
      OUT     W167.5
